FUNCTION_BLOCK FB_Estacion
VAR_INPUT
	
	// Variables de control
	EstadoPausa: BOOL;
	EstadoReinicia: BOOL;
	UnidadesSolicitadas: UINT := 3;
	TpoCintaDelSensorAlTope: TIME := T#400MS;
	TpoVerificador: TIME := T#2000MS;
	TpoDesplazador: TIME := T#400MS;
	TpoRechazador: TIME := T#500MS;
	TpoCintaFuera: TIME := T#2000MS;
	TpoRetenedorBaja: TIME := T#500MS;
	
END_VAR
VAR_OUTPUT
	
	// Parámetros
	CondicionInicial: BOOL;
	UnidadesPendientes: UINT;
	UnidadesRealizadas: UINT;
	
	// Entradas comunes
	PulsadorEmergencia AT %I*: BOOL;
    SelectorManual AT %I*: BOOL;
    PulsadorMarcha AT %I*: BOOL;
    PulsadorParada AT %I*: BOOL := TRUE; // Contacto normalmente cerrado
    EstacionConectada AT %I*: BOOL := TRUE;
    DetectorPresion AT %I*: BOOL := TRUE;
	
	PalePresencia AT %I*: BOOL;
    PaleCodigoBit0 AT %I*: BOOL;
    PaleCodigoBit1 AT %I*: BOOL;
    PaleCodigoBit2 AT %I*: BOOL;
	
	// Entradas específicas
	DescargadorDetras AT %I*: BOOL;
	DescargadorDelante AT %I*: BOOL;
	VerticalArriba AT %I*: BOOL;
	VerticalAbajo AT %I*: BOOL;
	VerificadorArriba AT %I*: BOOL;
	VerificadorAbajo AT %I*: BOOL;
	DesplazadorDetras AT %I*: BOOL;
	AlimentadorDetras AT %I*: BOOL;
	AlimentadorDelante AT %I*: BOOL;
	VacioDescargador AT %I*: BOOL;
	PresenciaBaseAlimentador AT %I*:BOOL;
END_VAR
VAR
	// Bloques funcionales
	Coordinador: FB_Coordinador_SFC;
	SituarBase: FB_1_SituarBase_SFC;
	AlimentarBase: FB_2_AlimentarBase_SFC;
	VerificarPale: FB_3_VerificarPale_SFC;
	InsertarBasePale: FB_4_InsertarBasePale_SFCC;
	TransferirBase: FB_5_TransferirBase_SFC;
	
	
	// Salidas comunes
	DesconectaEstacion AT %Q*: BOOL;
    LamparaAlarma AT %Q*: BOOL;
    LamparaMarcha AT %Q*: BOOL;
	LamparaFaltaMaterial AT %Q*: BOOL;
    AvisadorSonoro AT %Q*: BOOL;

    CintaMotorActiva AT %Q*: BOOL;
    CintaMotorInvierte AT %Q*: BOOL;
    CintaRetenedorBaja AT %Q*: BOOL;
    CintaSeparadorSube AT %Q*: BOOL;
	
	// Salidas específicas
	DescargadorAtras AT %Q*: BOOL;
	DescargadorAdelante AT %Q*: BOOL;
	DescargadorBaja AT %Q*: BOOL;
	RechazadorAdelante AT %Q*: BOOL;
	VerificadorBaja AT %Q*: BOOL;
	DesplazadorAdelante AT %Q*: BOOL;
	AlimentadorAdelante AT %Q*: BOOL;
	EyectorSucciona AT %Q*: BOOL;
END_VAR

// MODO AUTOMÁTICO
IF NOT SelectorManual THEN
	
//Bloques funcionales
Coordinador(
	UnidadesPendientes := UnidadesPendientes,
	UnidadesRealizadas := UnidadesRealizadas,
	SFCPause := NOT EstadoReinicia AND EstadoPausa,
	SFCReset := EstadoReinicia,
	Ack := TRUE,
	Execute := CondicionInicial AND (UnidadesSolicitadas > 0) AND PulsadorMarcha,
	BaseSituada := SituarBase.Done,
	PaleSituado := AlimentarBase.Done,
	PaleVerificado := VerificarPale.Done,
	PaleDesechado := VerificarPale.DoneIncorrecto,
	PaleTransferido := InsertarBasePale.Done,
	BaseSituada := TransferirBase.Done,
	CondicionInicial := CondicionInicial,
	UnidadesSolicitadas := UnidadesSolicitadas
);
	
SituarBase(
	SFCPause := NOT EstadoReinicia AND EstadoPausa,
	SFCReset := EstadoReinicia,
	Ack := NOT Coordinador.SituaBase,
	Execute := Coordinador.SituaBase,
	PalePresencia := PalePresencia,
	TpoCintaDelSensorAlTope := TpoCintaDelSensorAlTope,
);
	
AlimentarBase(
	SFCPause := NOT EstadoReinicia AND EstadoPausa,
	SFCReset := EstadoReinicia,
	Ack := NOT Coordinador.SituaPale,
	Execute := Coordinador.SituaPale,
	PresenciaBaseAlimentador := PresenciaBaseAlimentador,
	AlimentadorDelante := AlimentadorDelante,
	AlimentadorDetras := AlimentadorDetras,
);

VerificarPale(
	SFCPause := NOT EstadoReinicia AND EstadoPausa,
	SFCReset := EstadoReinicia,
	Ack := NOT Coordinador.VerificaPale,
	Execute := Coordinador.VerificaPale,
	VerificadorAbajo := VerificadorAbajo,
	VerificadorArriba := VerificadorArriba,
	DesplazadorDetras := DesplazadorDetras,
	TpoVerificador := TpoVerificador,
	TpoDesplazador := TpoDesplazador,
	TpoRechazador := TpoRechazador,	
);

InsertarBasePale(
	SFCPause := NOT EstadoReinicia AND EstadoPausa,
	SFCReset := EstadoReinicia,
	Ack := NOT Coordinador.TransfierePale,
	Execute := Coordinador.TransfierePale,
	VerticalAbajo := VerticalAbajo,
	VacioDescargador := VacioDescargador,
	VerticalArriba := VerticalArriba,
	DescargadorDelante := DescargadorDelante,
	DescargadorDetras := DescargadorDetras
);

TransferirBase(
	SFCPause := NOT EstadoReinicia AND EstadoPausa,
	SFCReset := EstadoReinicia,
	Ack := NOT Coordinador.TransfiereBase,
	Execute := Coordinador.TransfiereBase,
	TpoCintaFuera := TpoCintaFuera,
	TpoRetenedorBaja := TpoRetenedorBaja,
);

// Acciones

// DesconectaEstacion :=
LamparaAlarma := Coordinador.LamparaAlarma;
LamparaMarcha := Coordinador.LamparaMarcha;
// AvisadorSonoro :=

CintaMotorActiva := NOT EstadoPausa AND (SituarBase.CintaMotorActiva OR TransferirBase.CintaMotorActiva);
// CintaMotorInvierte :=
CintaRetenedorBaja := TransferirBase.CintaRetenedorBaja;
CintaSeparadorSube := TransferirBase.CintaSeparadorSube;
DescargadorAtras := InsertarBasePale.DescargadorAtras;
DescargadorAdelante := InsertarBasePale.DescargadorAdelante;
DescargadorBaja := InsertarBasePale.DescargadorBaja;
RechazadorAdelante := VerificarPale.RechazadorAdelante;
VerificadorBaja := VerificarPale.VerificadorBaja;
DesplazadorAdelante := VerificarPale.DesplazadorAdelante;
AlimentadorAdelante := AlimentarBase.AlimentadorAdelante;
EyectorSucciona := InsertarBasePale.EyectorSucciona;

END_IF

// Parámetros de salida
CondicionInicial := EstacionConectada AND AlimentadorDetras AND VerificadorArriba AND DesplazadorDetras AND DescargadorDetras AND VerticalArriba AND NOT VacioDescargador;

END_FUNCTION_BLOCK

(* stored: Version 1.1.0.1, ProductVersion 3.1.4024.12
   POU FB_Estacion: Id {3ae62a84-301f-41bd-b521-6369241fe03c}, SpecialFunc None *)
